{attribute 'qualified_only'}
{attribute 'strict'}
{attribute 'to_string'}
TYPE E_Steps :
(
	init := 0,
    enable,
    enabled,
    moveCenter,
    idle,
    enableExtSp,
    runExtSp,
    error
)UINT;
END_TYPE

(* stored: Version 1.1.0.1, ProductVersion 3.1.4026.18
   DUT E_Steps: Id {4fbc43e8-2a50-4b33-a22f-90e27858921c} *)
